DATA_BLOCK "Call_KeyenceCheckerIV_DB"
{ S7_Optimized_Access := 'TRUE' }
VERSION : 0.1
NON_RETAIN
"Call_KeyenceCheckerIV"

BEGIN

END_DATA_BLOCK

